FUNCTION_BLOCK FB_CauseNCError
VAR_IN_OUT
    Axis: AXIS_REF;
END_VAR
VAR_INPUT
    bExecute: BOOL;
    nErrorCode: UDINT;
END_VAR
VAR_OUTPUT
    bBusy: BOOL;
    bDone: BOOL;
END_VAR
VAR
    rtExec: R_TRIG;
    adsWrite: ADSWRITE;
    mcReadDriveAddress: MC_ReadDriveAddress;
END_VAR

rtExec(CLK:=bExecute);
IF NOT bExecute THEN
    bDone := FALSE;
END_IF
IF rtExec.Q THEN
    bBusy := TRUE;
END_IF
IF bBusy AND NOT mcReadDriveAddress.Done THEN
    mcReadDriveAddress(
        Axis:=Axis,
        Execute:=TRUE,
        DriveAddress=>Axis.DriveAddress);
END_IF
IF bBusy AND mcReadDriveAddress.Done THEN
    bBusy := TRUE;
    adsWrite(
        PORT:=501,
        IDXGRP:=16#4200 + Axis.DriveAddress.NcDriveId,
        IDXOFFS:=16#0019,
        LEN:=SIZEOF(nErrorCode),
        SRCADDR:=ADR(nErrorCode),
        WRITE:=TRUE,
        BUSY=>bBusy);
    IF NOT bBusy THEN
        bDone := TRUE;
        adsWrite(WRITE:=FALSE);
    END_IF
END_IF

END_FUNCTION_BLOCK

(* stored: Version 1.1.0.1, ProductVersion 3.1.4022.18
   POU FB_CauseNCError: Id {e3bbaf77-4a8b-41ac-91d3-26573b2f18e7}, SpecialFunc None *)
